VAR_GLOBAL CONSTANT
	iDoutputChannelCount : INT := 48;
END_VAR
VAR_GLOBAL
	bDigitalOut AT %Q*	: ARRAY [1..iDoutputChannelCount] OF BOOL;
	bDigitalOutFdbk : ARRAY [1..iDoutputChannelCount] OF BOOL;
	iDoutChannel	: ARRAY [1..iDoutputChannelCount] OF INT;
END_VAR

(* stored: Version 1.1.0.1, ProductVersion 3.1.4024.12
   GVL GVL_DigitalOut: Id {14e45cec-eb20-4b33-bf1e-8d96187f281c} *)
